Staubli VAL3: MotionCfgVel.pjx

--- MotionCfgVel.pjx ---
Parameters version=s7.8.1 stackSize=5000 millimeterUnit=true
Program file=start.pgx
Program file=stop.pgx
Data file=MotionCfgVel.dtx

--- MotionCfgVel.dtx ---
public frame fReference = {fatherId=world[0]}
public mdesc mMaxSpeed
public tool tTool = {fatherId=flange[0], ioLink=valve1}
public num nCmdType

--- stop.pgx ---
program stop()
begin
  // Copyright (c) 2021, Institute for Factory Automation and Production Systems (FAPS)
  //
  // Licensed under the Apache License, Version 2.0 (the "License");
  // you may not use this file except in compliance with the License.
  // You may obtain a copy of the License at
  //
  //     http://www.apache.org/licenses/LICENSE-2.0
  //
  // Unless required by applicable law or agreed to in writing, software
  // distributed under the License is distributed on an "AS IS" BASIS,
  // WITHOUT WARRANTIES OR CONDITIONS OF ANY KIND, either express or implied.
  // See the License for the specific language governing permissions and
  // limitations under the License.


end
